FUNCTION_BLOCK FB_TestFunction
VAR_INPUT
END_VAR
VAR_OUTPUT
END_VAR
VAR
END_VAR

END_FUNCTION_BLOCK

(* stored: Version 1.1.0.1, ProductVersion 3.1.4024.11
   POU FB_TestFunction: Id {202e3aee-003d-4ef2-8f26-aaa665cfe0a3}, SpecialFunc None *)
